// TIA Portal V16 program export: 1 tag tables, 0 data types, 0 data blocks, 5 code blocks (in call order from the OBs), 3 instance data blocks

VAR_GLOBAL   // PLC tag table "Standard-Variablentabelle"
   bool1 AT %I0.0 : Bool;
   bool2 AT %I0.1 : Bool;
END_VAR

ORGANIZATION_BLOCK "Main"   // OB1, LAD, ProgramCycle
TITLE = "Main Program Sweep (Cycle)"
VERSION : 0.1
// stored: IsIECCheckEnabled false
   VAR_TEMP
      OB1_EV_CLASS : Byte;   // Bits 0-3 = 1 (Coming event), Bits 4-7 = 1 (Event class 1)
      OB1_SCAN_1 : Byte;   // 1 (Cold restart scan 1 of OB 1), 3 (Scan 2-n of OB 1)
      OB1_PRIORITY : Byte;   // Priority of OB Execution
      OB1_OB_NUMBR : Byte;   // 1 (Organization block 1, OB1)
      OB1_RESERVED_1 : Byte;   // Reserved for system
      OB1_RESERVED_2 : Byte;   // Reserved for system
      OB1_PREV_CYCLE : Int;   // Cycle time of previous OB1 scan (milliseconds)
      OB1_MIN_CYCLE : Int;   // Minimum cycle time of OB1 (milliseconds)
      OB1_MAX_CYCLE : Int;   // Maximum cycle time of OB1 (milliseconds)
      OB1_DATE_TIME : Date_And_Time;   // Date and time OB1 started
   END_VAR
BEGIN

REGION Network 1
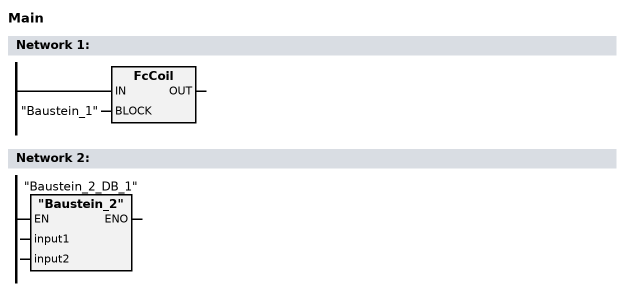
   // no SCL statement known for FcCoil: written as a call
   FcCoil(in := TRUE, block := "Baustein_1");
END_REGION

REGION Network 2
   RUNG wire#powerrail
      "Baustein_2_DB_1"(input1 :=, input2 :=)
   END_RUNG
   // the same network as SCL:
   "Baustein_2_DB_1"();   // "Baustein_2"
END_REGION
END_ORGANIZATION_BLOCK

FUNCTION_BLOCK "Baustein_2"   // FB2, STL
VERSION : 0.1
// stored: AutoNumber true, UDAEnableTagReadback false
   VAR_INPUT
      input1 : Bool;
      input2 : Bool;
   END_VAR
BEGIN

NETWORK
TITLE = 
      A     #input2;
      A     #input1;
      =     "bool2";



END_FUNCTION_BLOCK

ORGANIZATION_BLOCK "CYC_INT5_RTG1"   // OB35, LAD, CyclicInterrupt
TITLE = "Cyclic Interrupt"
VERSION : 0.1
// stored: IsIECCheckEnabled false
   VAR_TEMP
      OB35_EV_CLASS : Byte;   // Bits 0-3 = 1 (Coming event), Bits 4-7 = 1 (Event class 1)
      OB35_STRT_INF : Byte;   // 16#36 (OB 35 has started)
      OB35_PRIORITY : Byte;   // Priority of OB Execution
      OB35_OB_NUMBR : Byte;   // 35 (Organization block 35, OB35)
      OB35_RESERVED_1 : Byte;   // Reserved for system
      OB35_RESERVED_2 : Byte;   // Reserved for system
      OB35_PHASE_OFFSET : Word;   // Phase offset (msec)
      OB35_RESERVED_3 : Int;   // Reserved for system
      OB35_EXC_FREQ : Int;   // Frequency of execution (msec)
      OB35_DATE_TIME : Date_And_Time;   // Date and time OB35 started
   END_VAR
BEGIN

REGION Network 1
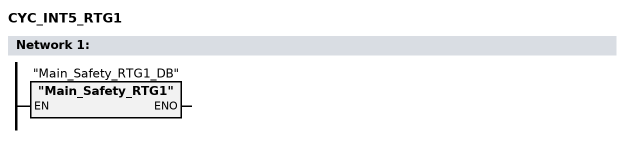
   RUNG wire#powerrail
      "Main_Safety_RTG1_DB"()
   END_RUNG
   // the same network as SCL:
   "Main_Safety_RTG1_DB"();   // "Main_Safety_RTG1"
END_REGION
END_ORGANIZATION_BLOCK

FUNCTION_BLOCK "Main_Safety_RTG1"   // FB1, F_LAD
VERSION : 0.1
// stored: AutoNumber false, IsIECCheckEnabled false, UDAEnableTagReadback false
BEGIN
END_FUNCTION_BLOCK

FUNCTION "Baustein_1" : Void   // FC1, FBD
VERSION : 0.1
// stored: AutoNumber true, IsIECCheckEnabled false, UDAEnableTagReadback false
BEGIN

REGION Network 1
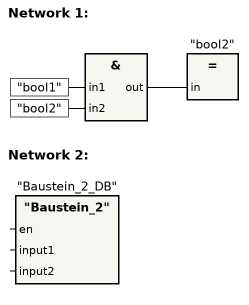
   "bool2" := "bool1" AND "bool2";
END_REGION

REGION Network 2
   "Baustein_2_DB"();   // "Baustein_2"
END_REGION
END_FUNCTION

DATA_BLOCK "Baustein_2_DB"   // DB2
VERSION : 0.1
// stored: AutoNumber true, InstanceOfName Baustein_2, InstanceOfType FB
"Baustein_2"
BEGIN
END_DATA_BLOCK

DATA_BLOCK "Baustein_2_DB_1"   // DB3
VERSION : 0.1
// stored: AutoNumber true, InstanceOfName Baustein_2, InstanceOfType FB
"Baustein_2"
BEGIN
END_DATA_BLOCK

DATA_BLOCK "Main_Safety_RTG1_DB"   // DB1, F_DB
VERSION : 0.1
// stored: AutoNumber false, InstanceOfName Main_Safety_RTG1, InstanceOfType FB
"Main_Safety_RTG1"
BEGIN
END_DATA_BLOCK
